{attribute 'qualified_only'}
VAR_GLOBAL CONSTANT
	MAX_HTTP_BODY_LENGTH 	: UDINT := 30000;
	MAX_HTTP_URL_LENGTH 	: UDINT := 1000;
END_VAR

(* stored: Version 1.1.0.1, ProductVersion 3.1.4020.3
   GVL GVL_HTTP_PARAMETERS: Id {fa0d35aa-5dcc-4507-964b-cdecc8beaba0} *)
